{attribute 'qualified_only'}
{attribute 'strict'}
TYPE E_DomeRotationState :
(
	idle  := 0,
	parked	:= 1,
	slewing := 2,
	error	:= 3,
	unknown := 4
);
END_TYPE

(* stored: Version 1.1.0.1, ProductVersion 3.1.4024.15
   DUT E_DomeRotationState: Id {c96709e9-bed9-4f1c-b47d-382f9c9b4e8c} *)
